(* calculate 16-bit checksum on a memory area *)
FUNCTION F_Checksum_CRC16 : WORD
VAR_INPUT
	bEnable		: BOOL;				(* TRUE = calculate checksum *)
	pSrcAddr	: POINTER TO BYTE;	(* pointer to 1st byte of memory area *)
	nBytes		: UDINT;			(* no of bytes to be included in checksum calculation *)
	nStartCRC	: UINT;				(* initial value used for checksum calculation *)
END_VAR
VAR
END_VAR
(*
-------------------------------------------------------------------------------------------------
Date		Version	Author	Comments
-------------------------------------------------------------------------------------------------
30/01/2015	3.00.00	PB		No change

-------------------------------------------------------------------------------------------------
05/02/10	1.00.00	PB		Initial release

-------------------------------------------------------------------------------------------------
*)

(* calculate checksum when bEnable = TRUE *)
IF bEnable = TRUE THEN

	F_Checksum_CRC16 := F_DATA_TO_CRC16_CCITT(pSrcAddr, nBytes, nStartCRC);
END_IF

END_FUNCTION

(* stored: Version 1.1.0.1
   POU F_Checksum_CRC16: Id {bbbb5561-0a50-47c8-af29-40538cc165e4}, SpecialFunc None *)
